// TwinCAT 3 PLC project HueControl
// ProgramVersion: 3.1.4023.0
// libraries:
//   Tc2_Standard, * (Beckhoff Automation GmbH)
//   Tc2_System, * (Beckhoff Automation GmbH)
//   Tc2_Utilities, * (Beckhoff Automation GmbH)
//   Tc3_IotBase, * (Beckhoff Automation GmbH)
//   Tc3_JsonXml, * (Beckhoff Automation GmbH)
//   Tc3_Module, * (Beckhoff Automation GmbH)
// project tree:
//   GVLs/ GVL.TcGVL
//   / PlcTask.TcTTO
//   POUs/ FB_TestHTTP_Put_PhilipsHue.TcPOU, MAIN.TcPOU
// real-time tasks:
//   TASK PlcTask: cycle T#10ms, priority 20, ADS port 350

CONFIGURATION HueControl
    RESOURCE PLC ON TwinCAT3
        TASK PlcTask(INTERVAL := T#10ms, PRIORITY := 20);
        PROGRAM MAIN WITH PlcTask : MAIN;
    END_RESOURCE
END_CONFIGURATION

// ---- GVLs/GVL.TcGVL
{attribute 'qualified_only'}
VAR_GLOBAL
	
	i32 : DINT;
END_VAR

// ---- POUs/MAIN.TcPOU
PROGRAM MAIN
VAR
	fbOpenFile		: FB_FileOpen;
	fbReadFile		: FB_FileRead;
	fbCloseFile		: FB_FileClose;

	
	fbOpenFile2		: FB_FileOpen;
	fbReadFile2		: FB_FileRead;
	fbCloseFile2	: FB_FileClose;
	
	workingPATH : STRING(84) := 'C:\Users\SamuelB\Documents\TcXaeShell\TwinCAT IOT\TwinCAT IOT\HueControl\POUs\Keys\';
	
	ADSRout : STRING(12);
	APIKey : STRING(40);
    // trigger command execution for Philips Hue samples
    bPutPhilipsHue : BOOL;

    fbHttpClientPhilipsHue         : FB_IotHttpClient :=(bKeepAlive:=TRUE, tConnectionTimeout:=T#10S);

    fbHttpPutPhilipsHue            : FB_TestHTTP_Put_PhilipsHue;

    bBlinkingMode                  : BOOL;
    fbTimer                        : TON:=(PT:=T#1MS);
    nColor                         : UINT;

	nBrightness: UINT := 100;
	nSaturation: UINT := 200;
	
	x : LREAL;
	y : LREAL;
	
	xy : ARRAY[0..1] OF LREAL;
	nState: INT;
END_VAR

CASE nState OF
	
	0:
		fbOpenFile.bExecute := TRUE;
		nState := 1;

	1:
		fbOpenFile(
			sNetId:= '', 
			sPathName:= CONCAT(workingPATH, 'ads.config'), 
			nMode:= FOPEN_MODEREAD);
			
		IF NOT fbOpenFile.bError AND NOT fbOpenFile.bBusy THEN
			fbOpenFile.bExecute := FALSE;
			fbReadFile.bExecute := TRUE;
			nState := 2;
		END_IF
		
	2:
		fbReadFile(
			sNetId:= '', 
			hFile:= fbOpenFile.hFile, 
			pReadBuff:= ADR(ADSRout), 
			cbReadLen:= SIZEOF(ADSRout));
			
		IF NOT fbReadFile.bBusy AND NOT fbReadFile.bError THEN
			fbReadFile.bExecute := FALSE;
			fbCloseFile.bExecute := TRUE;
			nState := 3;
		END_IF

	3:
		fbCloseFile(
			sNetId:= '', 
			hFile:= fbReadFile.hFile);
			
		IF NOT fbCloseFile.bBusy AND NOT fbCloseFile.bError THEN
			fbCloseFile.bExecute := FALSE;
			fbOpenFile2.bExecute := TRUE;
			nState := 4;
		END_IF
		
	4:
		fbOpenFile2(
			sNetId:= '', 
			sPathName:= CONCAT(workingPATH, 'apiKey.config'), 
			nMode:= FOPEN_MODEREAD);
			
		IF NOT fbOpenFile2.bError AND NOT fbOpenFile2.bBusy THEN
			fbOpenFile2.bExecute := FALSE;
			fbReadFile2.bExecute := TRUE;
			nState := 5;
		END_IF
		
	5:
		fbReadFile2(
			sNetId:= '', 
			hFile:= fbOpenFile2.hFile, 
			pReadBuff:= ADR(APIKey), 
			cbReadLen:= SIZEOF(APIKey));
			
		IF NOT fbReadFile2.bBusy AND NOT fbReadFile2.bError THEN
			fbReadFile2.bExecute := FALSE;
			fbCloseFile2.bExecute := TRUE;
			nState := 6;
		END_IF

	6:
		fbCloseFile2(
			sNetId:= '', 
			hFile:= fbReadFile2.hFile);
			
		IF NOT fbCloseFile2.bBusy AND NOT fbCloseFile2.bError THEN
			fbCloseFile2.bExecute := FALSE;
			nState := 7;
		END_IF
		
	7:
		fbHttpClientPhilipsHue.sHostName := ADSRout;
		nState := 8;
		
		
	8:
		//init client parameters at startup
		xy[0] := x;
		xy[1] := y;
		
		IF NOT fbHttpClientPhilipsHue.bConfigured THEN
			fbHttpClientPhilipsHue.nHostPort:= 80;
			fbHttpClientPhilipsHue.stTLS.bNoServerCertCheck:= FALSE;
		END_IF
		
		IF fbHttpClientPhilipsHue.bConfigured THEN
			fbHttpPutPhilipsHue(bSend:=bPutPhilipsHue, fbClient:=fbHttpClientPhilipsHue, xy := xy, nBrightness := nBrightness, APIKey := APIKey);
		END_IF
		
		IF bBlinkingMode THEN
			fbTimer(IN:=NOT fbTimer.Q);
			IF fbTimer.Q THEN
				IF bPutPhilipsHue THEN
					bPutPhilipsHue:=FALSE;
				ELSE
					bPutPhilipsHue:=TRUE;
				END_IF
			END_IF
		END_IF
		
		fbHttpClientPhilipsHue.Execute();
	
END_CASE

END_PROGRAM

// ---- POUs/FB_TestHTTP_Put_PhilipsHue.TcPOU
FUNCTION_BLOCK FB_TestHTTP_Put_PhilipsHue
VAR_INPUT
	    bSend                : BOOL;
		xy					 : ARRAY[0..1] OF LREAL;
		nBrightness			 : UINT;
		APIKey				 : STRING(40);
END_VAR
VAR_IN_OUT
		fbClient             : FB_IotHttpClient;
END_VAR
VAR_OUTPUT
		bBusy                : BOOL;
    	bError               : BOOL;
END_VAR
VAR
	fbRequest            : FB_IotHttpRequest;
    fbJson               : FB_JsonDomParser;
    fbJsonWriter         : FB_JsonSaxWriter;
    nState               : UDINT;
    RisingEdge           : R_TRIG;
    
    bGetContentResult    : BOOL;
    sContent             : STRING(511);
    sSend                : STRING(511);
    
    bGetJsonResult       : BOOL;
    jsonDoc              : SJsonValue;
    jsonVal              : SJsonValue;
    sResultValue         : STRING;
    
    nReqCount            : UDINT;    
    nResCount            : UDINT;
    nValidResCount       : UDINT;
    nErrCount            : UDINT;
    
    fbTimer              : TON;
    bLightOn             : BOOL;
	sURIPath: STRING(255);
END_VAR

RisingEdge(CLK:= bSend );

sURIPath := CONCAT('/api/',CONCAT(APIKey,'/lights/1/state'));

CASE nState OF
0:    
        fbJsonWriter.StartObject();
        fbJsonWriter.AddKey('on');
        fbJsonWriter.AddBool(TRUE);
        fbJsonWriter.AddKey('bri');
        fbJsonWriter.AddUdint(nBrightness);
		fbJsonWriter.AddKey('xy');
		fbJsonWriter.StartArray();
		fbJsonWriter.AddLReal(xy[0]);
		fbJsonWriter.AddLReal(xy[1]);
		fbJsonWriter.EndArray();
        fbJsonWriter.EndObject();
		
		
        sSend:=fbJsonWriter.GetDocument();
        fbJsonWriter.ResetDocument();
    IF RisingEdge.Q THEN 
        IF fbRequest.SendRequest(sUri:= sURIPath, fbClient:=fbClient, eRequestType:=ETcIotHttpRequestType.HTTP_PUT, 
            pContent:=ADR(sSend), nContentSize:=LEN2(ADR(sSend)), 0) THEN                
            nState:= 1;
            nReqCount:= nReqCount+1;
            bBusy:= TRUE;
            bError:= FALSE;
        END_IF                    
    END_IF
1:
    IF NOT fbRequest.bBusy THEN
        bError:= TRUE;
        IF NOT fbRequest.bError THEN                 
            bGetContentResult:= fbRequest.GetContent(pContent:= ADR(sContent), nContentSize:= SIZEOF(sContent), bSetNullTermination:= TRUE);
            IF fbRequest.nStatusCode >= 200 AND fbRequest.nStatusCode < 300 THEN
                bGetJsonResult:= FALSE;
                jsonDoc:= fbRequest.GetJsonDomContent(fbJson);
                IF jsonDoc <> 0 THEN
                    ; // do something with status response
                    nValidResCount:= nValidResCount+1;
                    bError:= FALSE;    
                END_IF                            
                nResCount:= nResCount+1;            
            END_IF
        END_IF
        nState:= 0;
        bBusy:= FALSE;
        IF bError THEN
            nErrCount:= nErrCount+1;
        END_IF
    END_IF      
END_CASE

END_FUNCTION_BLOCK
